{attribute 'qualified_only'}
VAR_GLOBAL
    {attribute 'pytmc' := 'pv: PLC:TXI:SXR:MOTION:ARB:01'}
    fbArbiter1: FB_Arbiter(1);

    // For all devices after Stopper
    {attribute 'pytmc' := 'pv: PLC:TXI:SXR:MOTION:FFO:01'}
    {attribute 'TcLinkTo' := '.q_xFastFaultOut:=TIIB[PMPS_FFO]^Channel 1^Output'}
    fbFastFaultOutput1: FB_HardwareFFOutput := (bAutoReset := TRUE, i_sNetID:='');

     {attribute 'pytmc' := 'pv: PLC:TXI:K:MOTION:PMPS:ReqTrans'}
    rReqTrans AT %I*		: ARRAY [1..PMPS_GVL.AUX_ATTENUATORS] OF ST_PMPS_Attenuator_IO;
    {attribute 'pytmc' := 'pv: PLC:TXI:K:MOTION:PMPS:CurTrans'}
    rCurTrans AT %Q*		: ARRAY [1..PMPS_GVL.AUX_ATTENUATORS] OF ST_PMPS_Attenuator_IO;


END_VAR

(* stored: Version 1.1.0.1
   GVL GVL: Id {a78c9729-a980-0963-1a01-5fb12e0c24b3} *)
